PROGRAM MAIN
VAR
	i : INT;
END_VAR

i := i + 1;

IpcDiagnostics();		// first way to implement the IPC diagnostics

//IpcDiagnostics_2();		// second way to implement the IPC diagnostics

END_PROGRAM

(* stored: Version 1.1.0.1, ProductVersion 3.1.4022.18
   POU MAIN: Id {ebf68f6f-cb24-4b94-876b-484c15003446}, SpecialFunc None *)
